// SIMATIC S7-200 SMART project (STEP 7-Micro/WIN SMART), CPU SR40

ORGANIZATION_BLOCK MAIN:OB1
TITLE=程序注释
BEGIN
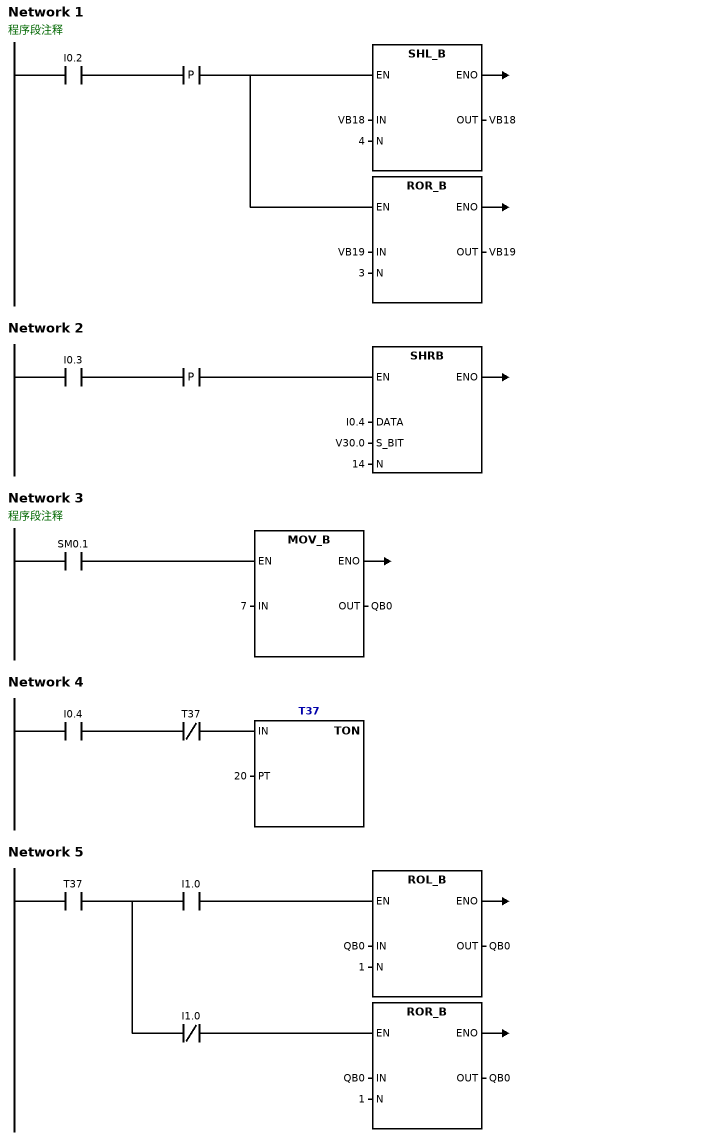
Network 1
// 程序段注释
LD     I0.2
EU
SLB    VB18, 4
RRB    VB19, 3
Network 2
LD     I0.3
EU
SHRB   I0.4, V30.0, 14
Network 3
// 程序段注释
// (network saved uncompiled; LAD cells follow)
// row 0: c0 -| |- SM0.1  c1 --  c2 [MOV_B EN:=power@row0, IN:=7, ENO=>power, OUT=>QB0]  c3 ->
// row 1: c2 [box]
Network 4
// (network saved uncompiled; LAD cells follow)
// row 0: c0 -| |- I0.4  c1 -|/|- T37  c2 [TON T37 IN:=power@row0, PT:=20]
// row 1: c2 [box]
Network 5
LD     T37
LPS
A      I1.0
RLB    QB0, 1
LPP
AN     I1.0
RRB    QB0, 1
END_ORGANIZATION_BLOCK
